// Mitsubishi GX Works2 project: lights   PLC: FX1S

PROGRAM MAIN
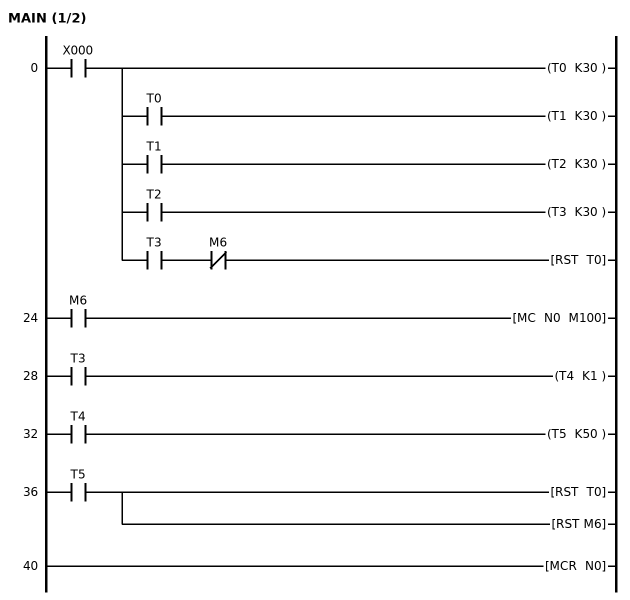
0     LD      X000
      OUT     T0 K30
      MPS
      AND     T0
      OUT     T1 K30
      MRD
      AND     T1
      OUT     T2 K30
      MRD
      AND     T2
      OUT     T3 K30
      MPP
      AND     T3
      ANI     M6
      RST     T0
24    LD      M6
      MC      N0 M100
28    LD      T3
      OUT     T4 K1
32    LD      T4
      OUT     T5 K50
36    LD      T5
      RST     T0
      RST     M6
40    MCR     N0
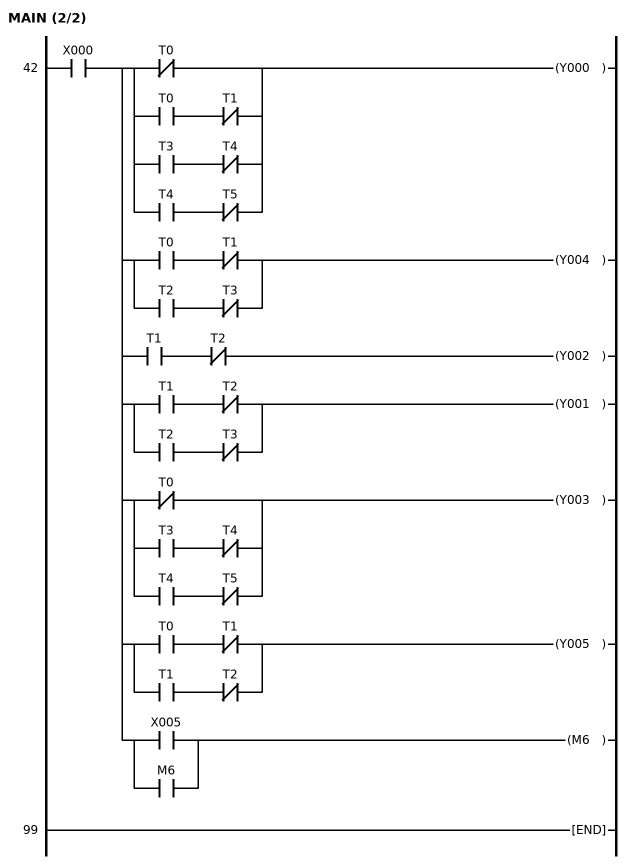
42    LD      X000
      MPS
      LDI     T0
      LD      T0
      ANI     T1
      ORB
      LD      T3
      ANI     T4
      ORB
      LD      T4
      ANI     T5
      ORB
      ANB
      OUT     Y000
      MRD
      LD      T0
      ANI     T1
      LD      T2
      ANI     T3
      ORB
      ANB
      OUT     Y004
      MRD
      AND     T1
      ANI     T2
      OUT     Y002
      MRD
      LD      T1
      ANI     T2
      LD      T2
      ANI     T3
      ORB
      ANB
      OUT     Y001
      MRD
      LDI     T0
      LD      T3
      ANI     T4
      ORB
      LD      T4
      ANI     T5
      ORB
      ANB
      OUT     Y003
      MRD
      LD      T0
      ANI     T1
      LD      T1
      ANI     T2
      ORB
      ANB
      OUT     Y005
      MPP
      LD      X005
      OR      M6
      ANB
      OUT     M6
99    END
END_PROGRAM
